// TwinCAT 3 PLC project PLC1
// Title: CoffeeMaker
// Company: Brandon
// ProjectVersion: 0.1
// ProgramVersion: 3.1.4026.21
// libraries:
//   SPT Base Types, * (Beckhoff Automation LLC)
//   Tc2_Standard, * (Beckhoff Automation GmbH)
//   Tc2_System, * (Beckhoff Automation GmbH)
// project tree:
//   Component/FBs/ FB_HeatingElement.TcPOU, FB_SimulatedPump.TcPOU, FB_SimulatedScale.TcPOU, FB_SimulatedTempSensor.TcPOU
//   Component/Interfaces/ I_HeatingElement.TcIO, I_Pump.TcIO (not stored), I_Scale.TcIO (not stored), I_TempSensor.TcIO
//   Equipment/FBs/ FB_Boiler.TcPOU, FB_Dispenser.TcPOU
//   Equipment/Interfaces/ I_Boiler.TcIO (not stored), I_Dispenser.TcIO (not stored)
//   Machine/ FB_Machine.TcPOU
//   / MAIN.TcPOU, PlcTask.TcTTO
//   Misc/LinkedList/ FB_LinkedList.TcPOU, F_Copy_Generic.TcPOU (not stored), POU.TcPOU, ST_Node.TcDUT, T_Generic.TcDUT
//   _DUTs/ENUMs/ E_State.TcDUT
// real-time tasks:
//   TASK PlcTask: cycle T#10ms, priority 20, ADS port 350
//   TASK PlcTask1: cycle T#10ms, priority 21, ADS port 351

CONFIGURATION PLC1
    RESOURCE PLC ON TwinCAT3
        TASK PlcTask(INTERVAL := T#10ms, PRIORITY := 20);
        PROGRAM MAIN WITH PlcTask : MAIN;
    END_RESOURCE
END_CONFIGURATION

// ---- Misc/LinkedList/ST_Node.TcDUT
{attribute 'enable_dynamic_creation'}
TYPE ST_Node :
STRUCT
	data : T_Generic;
	pNext : POINTER TO INT;
	pPrev : POINTER TO INT;
END_STRUCT
END_TYPE

// ---- Misc/LinkedList/T_Generic.TcDUT
TYPE T_Generic : __SYSTEM.AnyType ; END_TYPE

// ---- _DUTs/ENUMs/E_State.TcDUT
//{attribute 'qualified_only'}
{attribute 'strict'}
{attribute 'to_string'}
TYPE E_State :
(
	IDLE,
	STARTING,
	EXECUTE,
	HOLDING,
	UNHOLDING,
	HELD,
	COMPLETING,
	COMPLETED,
	RESETTING,
	ABORTING,
	ABORTED,
	CLEARING,
	STOPPING,
	STOPPED	
);
END_TYPE

// ---- Component/Interfaces/I_HeatingElement.TcIO
INTERFACE I_HeatingElement EXTENDS I_ComponentBase

METHOD Disable
VAR_INPUT
END_VAR
END_METHOD

METHOD Enable
VAR_INPUT
END_VAR
END_METHOD

METHOD Init
VAR_INPUT
END_VAR
END_METHOD

PROPERTY isHeating : BOOL
GET
END_GET
END_PROPERTY

METHOD PowerOff : BOOL
VAR_INPUT
END_VAR
END_METHOD

METHOD PowerOn : BOOL
VAR_INPUT
END_VAR
END_METHOD

PROPERTY State : E_State
GET
END_GET
END_PROPERTY

END_INTERFACE

// ---- Component/Interfaces/I_TempSensor.TcIO
INTERFACE I_TempSensor EXTENDS I_ComponentBase

PROPERTY SimulatedHeatingElement : I_HeatingElement
GET
END_GET
SET
END_SET
END_PROPERTY

PROPERTY Temp : LREAL
GET
END_GET
END_PROPERTY

END_INTERFACE

// ---- MAIN.TcPOU
PROGRAM MAIN
VAR
END_VAR

END_PROGRAM

// ---- Component/FBs/FB_HeatingElement.TcPOU
FUNCTION_BLOCK FB_HeatingElement EXTENDS FB_ComponentBase IMPLEMENTS I_HeatingElement
VAR
	_enabled 	: BOOL;				
	_output  	AT %Q* : BOOL;
	_state		: E_State := ABORTED;
END_VAR

///////////////////////////////////////////////////////////////////////////////////////////
//
//	States:
//	Before initializing: ABORTED
//	Once initialized, disabled: STOPPED
//	Once initialized, enabled: IDLE
//	Once enabled, PowerOn: EXECUTE
//	Once enabled, PowerOff: IDLE
//
//
//

METHOD Disable
_enabled := FALSE;
PowerOff();
_State := STOPPED;
END_METHOD

METHOD Enable
_enabled := TRUE;
_State := IDLE;
END_METHOD

METHOD Init
_enabled := FALSE;
PowerOff();
_State := STOPPED;
END_METHOD

PROPERTY isHeating : BOOL
GET
isHeating := _output;
END_GET
END_PROPERTY

METHOD PowerOff : BOOL
_output := FALSE;
_State := IDLE;
END_METHOD

METHOD PowerOn : BOOL
IF _enabled THEN
	_output := TRUE;
	_State := EXECUTE;
END_IF
END_METHOD

PROPERTY State : E_State
GET
END_GET
END_PROPERTY

END_FUNCTION_BLOCK

// ---- Component/FBs/FB_SimulatedPump.TcPOU
FUNCTION_BLOCK FB_SimulatedPump EXTENDS FB_ComponentBase IMPLEMENTS I_Pump
VAR_INPUT
END_VAR
VAR_OUTPUT
END_VAR
VAR
END_VAR

{warning 'Add method implementation '}
METHOD CyclicLogic
END_METHOD

{warning 'Add property implementation'}
PROPERTY Speed : LREAL
GET
END_GET
SET
END_SET
END_PROPERTY

{warning 'Add method implementation '}
METHOD Start : BOOL
END_METHOD

{warning 'Add method implementation '}
METHOD Stop
END_METHOD

END_FUNCTION_BLOCK

// ---- Component/FBs/FB_SimulatedScale.TcPOU
FUNCTION_BLOCK FB_SimulatedScale EXTENDS FB_ComponentBase IMPLEMENTS I_Scale
VAR_INPUT
END_VAR
VAR_OUTPUT
END_VAR
VAR
END_VAR

{warning 'Add method implementation '}
METHOD CyclicLogic
END_METHOD

{warning 'Add method implementation '}
METHOD Tare
END_METHOD

{warning 'Add property implementation'}
PROPERTY Weight : LREAL
GET
END_GET
SET
END_SET
END_PROPERTY

END_FUNCTION_BLOCK

// ---- Component/FBs/FB_SimulatedTempSensor.TcPOU
FUNCTION_BLOCK FB_SimulatedTempSensor EXTENDS FB_ComponentBase IMPLEMENTS I_TempSensor
VAR
	_SimulatedHeatingElement: I_HeatingElement;
	_Temp: LREAL := 20;
END_VAR

//{warning 'Add method implementation '}
METHOD CyclicLogic
VAR
	P_elec			: LREAL;			// Electric power for the heater (W)
	k_hw			: LREAL := 65;		// Heater --> Water coupling (W/deg C)
	h_h				: LREAL := 2;		// Heater --> air loss (W/deg C)
	T_ambient		: LREAL := 20;		// Room temperature (deg C)
	m_h				: LREAL := 0.22;	// Mass of the heater (kg)
	c_h				: LREAL := 500;		// Specific heat of heater (J/kg)
	delta_t 		: LREAL := 0.25;		// Change in time per cycle (s)
	h_w				: LREAL := 18;		// Water --> air loss (W/deg C)
	m_w				: LREAL := 0.75;		// Mass of the water (kg)
	c_w				: LREAL := 4180;	// Specific heat of water (J/kg)
END_VAR
VAR_INST
	T_h : LREAL := 20;
	T_w : LREAL := 20;
END_VAR
IF _SimulatedHeatingElement <> 0 THEN
	// Electrical Input
	P_elec := SEL(_SimulatedHeatingElement.isHeating, 0, 1000);
	// Heater Dynamics
	T_h := T_h + ((P_elec - k_hw * (T_h - T_w) - h_h * (T_h - T_ambient)) / (m_h * c_h)) * delta_t;
	// Water Dynamics
	T_w := T_w + ((k_hw * (T_h -T_w) - h_w * (T_w - T_ambient)) / (m_w * c_w)) *delta_t;
	IF T_w > 100 THEN
		T_w := 100;
	END_IF
	
	_Temp := T_w;
END_IF
END_METHOD

PROPERTY SimulatedHeatingElement : I_HeatingElement
GET
SimulatedHeatingElement := _SimulatedHeatingElement;
END_GET
SET
_SimulatedHeatingElement := SimulatedHeatingElement;
END_SET
END_PROPERTY

{warning 'Add property implementation'}
PROPERTY Temp : LREAL
GET
Temp := _Temp;
END_GET
END_PROPERTY

END_FUNCTION_BLOCK

// ---- Equipment/FBs/FB_Boiler.TcPOU
FUNCTION_BLOCK FB_Boiler EXTENDS FB_PackML_BaseModule IMPLEMENTS I_Boiler
VAR

END_VAR

PROPERTY CurrentTemp : LREAL
GET
IF ipTempSensor <> 0 THEN
	CurrentTemp := ipTempSensor.Temp;
END_IF
END_GET
END_PROPERTY

//{warning 'Add method implementation '}
METHOD CyclicLogic
VAR
END_VAR
IF _SimulateComponents THEN
	ipHeatingElement := Sim_Heater;
	ipTempSensor := Sim_TempSensor;
	ipTempSensor.SimulatedHeatingElement := ipHeatingElement;
END_IF

IF ipTempSensor <> 0 AND ipHeatingElement <> 0 THEN
	IF ipTempSensor.Temp < _TemperatureSetpoint THEN
		ipHeatingElement.PowerOn();
		_Heating := TRUE;
	ELSE
		ipHeatingElement.PowerOff();
		_Heating := FALSE;
	END_IF
	ipTempSensor.CyclicLogic();
	ipHeatingElement.CyclicLogic();
END_IF
END_METHOD

{warning 'Add method implementation '}
METHOD Disable : BOOL
END_METHOD

{warning 'Add method implementation '}
METHOD Enable : BOOL
END_METHOD

PROPERTY Heating : BOOL
GET
Heating := _Heating;
END_GET
END_PROPERTY

{warning 'Add property implementation'}
PROPERTY SetpointMet : BOOL
GET
END_GET
END_PROPERTY

PROPERTY SimulateComponents : BOOL
GET
SimulateComponents := _SimulateComponents;
END_GET
SET
_SimulateComponents := SimulateComponents;
END_SET
END_PROPERTY

{warning 'Add property implementation'}
PROPERTY TemperatureSetpoint : LREAL
GET
END_GET
SET
END_SET
END_PROPERTY

END_FUNCTION_BLOCK

// ---- Equipment/FBs/FB_Dispenser.TcPOU
FUNCTION_BLOCK FB_Dispenser EXTENDS FB_PackML_BaseModule IMPLEMENTS I_Dispenser
VAR
	// Interfaces
	ipPump	:	I_Pump;
	ipScale	:	I_Scale;
	
	// FBs
	DcPump		: FB_DcPump;
	SerialScale	: FB_SerialScale;
END_VAR

{warning 'Add method implementation '}
METHOD ChangeMode
VAR_INPUT
	Mode	: SPT_BaseTypes.E_PMLUnitMode;
END_VAR
END_METHOD

{warning 'Add method implementation '}
METHOD ChangeState
VAR_INPUT
	State	: SPT_BaseTypes.E_PMLCommand;
END_VAR
END_METHOD

{error 'Add property implementation or delete property to use base implementation'}
PROPERTY CurrentMode : SPT_BaseTypes.E_PMLUnitMode
GET
END_GET
END_PROPERTY

{error 'Add property implementation or delete property to use base implementation'}
PROPERTY CurrentState : SPT_BaseTypes.E_PMLState
GET
END_GET
END_PROPERTY

{warning 'Add method implementation '}
METHOD CyclicLogic
END_METHOD

{warning 'Add property implementation'}
PROPERTY Dispensing : BOOL
GET
END_GET
END_PROPERTY

{warning 'Add property implementation'}
PROPERTY Done : BOOL
GET
END_GET
END_PROPERTY

{warning 'Add method implementation '}
METHOD StartDispense
END_METHOD

METHOD Stop
END_METHOD

{warning 'Add property implementation'}
PROPERTY TargetWeight : LREAL
GET
END_GET
SET
END_SET
END_PROPERTY

END_FUNCTION_BLOCK

// ---- Machine/FB_Machine.TcPOU
FUNCTION_BLOCK FB_Machine EXTENDS FB_PackML_BaseModule
VAR
	Boiler		: 	I_Boiler;
	Dispenser	: 	I_Dispenser;
END_VAR

{warning 'Add method implementation '}
METHOD CyclicLogic
END_METHOD

END_FUNCTION_BLOCK

// ---- Misc/LinkedList/FB_LinkedList.TcPOU
FUNCTION_BLOCK FB_LinkedList
VAR
	pHead  : POINTER TO ST_Node;
	pTail  : POINTER TO ST_Node;
	Count  : UINT := 0; 
	
	pLastAccessed : POINTER TO ST_Node;
END_VAR

METHOD addValue
VAR_INPUT
	data : ANY;
END_VAR
VAR
	pTemp : POINTER TO ST_Node;
	pNode : POINTER TO ST_Node;
END_VAR
// Create a new node
pNode := __NEW(ST_Node, 1);
IF pNode <> 0 THEN
	// Give new node the input data
	pNode^.data := data;
	IF pHead = 0 THEN
		// List is currently empty, assign new node to head
		pHead := pNode;
		pTail := pNode;
	ELSIF Count = 1 THEN
		pHead^.pNext := pNode;
		pTail := pNode;
		pTail^.pPrev := pHead;
	ELSE
		pTemp := pTail;
		pTail := pNode;
		pTail^.pPrev :=pTemp;
		pTemp^.pNext := pTail;
	END_IF
	count := count + 1;
ELSE
	RETURN;
END_IF
END_METHOD

//FB_Exit must be implemented explicitly. If there is an implementation, then the
//method is called before the controller removes the code of the function block instance
//(implicit call). The return value is not evaluated.
METHOD FB_Exit: BOOL
VAR_INPUT
    bInCopyCode: BOOL;  // TRUE: the exit method is called in order to leave the instance which will be copied afterwards (online change).  

END_VAR
VAR
	i : UINT;
	pNext : POINTER TO ST_Node;
	pNode : POINTER TO ST_Node;
END_VAR
IF Count > 0 THEN
	pNode := pHead;
	
	IF Count = 1 THEN
		pNode^.pNext := 0;
		pNode^.pPrev := 0;
		__DELETE(pNode);
	ELSE
		FOR i := 0 TO Count-1 DO
			IF pNode <> pTail THEN
				pNext := pNode^.pNext;
			END_IF
			pNode^.pNext := 0;
			pNode^.pPrev := 0;
			__DELETE(pNode);
			pNode := pNext;
		END_FOR
	END_IF
END_IF
END_METHOD

//FB_Init is always available implicitly and it is used primarily for initialization.
//The return value is not evaluated. For a specific influence, you can also declare the
//methods explicitly and provide additional code there with the standard initialization
//code. You can evaluate the return value.
METHOD FB_Init: BOOL
VAR_INPUT
    bInitRetains: BOOL; // TRUE: the retain variables are initialized (reset warm / reset cold)
    bInCopyCode: BOOL;  // TRUE: the instance will be copied to the copy code afterward (online change)   
END_VAR
pHead := pTail := 0;
Count := 0;
END_METHOD

METHOD PRIVATE getNode : POINTER TO ST_Node
VAR_INPUT
	index : UINT;
END_VAR

VAR
	pNode : POINTER TO ST_Node;
	i: UINT;
END_VAR
pNode := pHead;
IF index >= 0 AND index < Count AND pNode <> 0 THEN 
	FOR i := 0 TO Count - 1 DO
		IF i = index THEN
			getNode := pNode;
			
			RETURN;
		END_IF
		pNode := pNode^.pNext;
	END_FOR
ELSE
	RETURN;
END_IF
END_METHOD

METHOD getValue
VAR_INPUT
	index : UINT;
	value : ANY;
END_VAR

VAR
	pNode : POINTER TO ST_Node;
	i: UINT;
END_VAR
pNode := getNode(index);
F_Copy_Generic(Source := pNode^.Data, Destination := Value);
END_METHOD

METHOD insertAfter : BOOL
VAR_INPUT
	value : ANY;
	position : UINT;
END_VAR
addValue(value);
moveAfter(count-1, position);
END_METHOD

METHOD isEmpty : BOOL
VAR_INPUT
END_VAR
isEmpty := Count = 0;
END_METHOD

PROPERTY Length : UINT
GET
Length := count;
END_GET
END_PROPERTY

METHOD MoveAfter : BOOL
VAR_INPUT
	MoveIndex : UINT;
	AfterIndex  : UINT;
END_VAR
VAR
	pMove : POINTER TO ST_Node;
	pAfter : POINTER TO ST_Node;
	
	pTemp : POINTER TO ST_Node;
END_VAR
pMove := getNode(MoveIndex);
pAfter:= getNode(AfterIndex);

// Check pointers are valid
IF pMove = 0 OR pAfter = 0 THEN
	RETURN;
END_IF

// No change needed
IF pMove = pAfter OR pAfter^.pNext = pMove THEN
	RETURN;
END_IF


// detach pMove
IF pMove^.pPrev <> 0 THEN
	pTemp := pMove^.pPrev;
	pTemp^.pNext := pMove^.pNext;
ELSE
	pHead := pMove^.pNext;
END_IF

IF pMove^.pNext <> 0 THEN
	pTemp := pMove^.pNext;
	pTemp^.pPrev := pMove^.pPrev;
ELSE 
	pTail := pMove^.pPrev;
END_IF

// insert after 
pMove^.pPrev := pAfter;
pMove^.pNext := pAfter^.pNext;

IF pAfter^.pNext <> 0 THEN
	pTemp := pAfter^.pNext;
	pTemp^.pPrev := pMove;
ELSE
	pTail := pMove;
END_IF

pAfter^.pNext := pMove;
END_METHOD

METHOD remove : BOOL
VAR_INPUT
	index : UINT;
END_VAR
VAR
	pNode : POINTER TO ST_Node;
	pPrevNode : POINTER TO ST_Node;
	pNextNode : POINTER TO ST_Node;
END_VAR
pNode := getNode(index);
pPrevNode := pNode^.pPrev;
pNextNode := pNode^.pNext;

pPrevNode^.pNext := pNextNode;
pNextNode^.pPrev := pPrevNode;

__DELETE(pNode);
count := count - 1;
END_METHOD

END_FUNCTION_BLOCK

// ---- Misc/LinkedList/POU.TcPOU
FUNCTION F_Copy_Generic : BOOL
VAR_INPUT
	Source, Destination : REFERENCE TO T_Generic;
END_VAR
VAR
	bSuccess : BOOL;
END_VAR

IF NOT (__ISVALIDREF(Source) OR_ELSE __ISVALIDREF(Destination)) THEN
	F_Copy_Generic := FALSE;
	RETURN;
END_IF

bSuccess := MEMCPY(Destination.pValue, Source.pValue, TO_UDINT(MIN(Source.diSize, Destination.diSize))) > 0;
F_Copy_Generic := bSuccess;

END_FUNCTION
